// TIA Portal V21 export
DATA_BLOCK "Trafiklys_DB"   // DB3
// stored: InstanceOfName Trafiklys, InstanceOfType FB
"Trafiklys"
   // VAR_INPUT
   //    i_start : Bool;
   //    i_suspendResume : Bool;
   //    i_manualMode : Bool;
   //    i_pushButtonEmergencyStop : Bool;
   //    i_manualRed : Bool;
   //    i_manualYellow : Bool;
   //    i_manualGreen : Bool;
   // END_VAR
   // VAR_OUTPUT
   //    o_red : Bool;
   //    o_yellow : Bool;
   //    o_green : Bool;
   // END_VAR
   // VAR
   //    statG0_step : Array[100..102] of Bool;
   //    statG1_step : Array[0..4] of Bool;
   //    statG2_step : Array[200..201] of Bool;
   //    statG3_step : Array[300..301] of Bool;
   //    statGManual : Array[5..5] of Bool;
   //    statSuspendResumeTrigger : R_TRIG;
   //    statTime { S7_SetPoint := 'True'} : Time;
   //    statTimer_G1_step : Array[1..4] of IEC_TIMER;
   // END_VAR
BEGIN
END_DATA_BLOCK
